// TIA Portal V17 export
// export: Created 2026-04-13T11:12:41.8044851Z, ExportSetting WithDefaults, DisplayName Totally Integrated Automation Portal, DisplayVersion V17 Update 4, DisplayName TIA Portal Openness, DisplayVersion V17 Update 4, DisplayName TIA Portal Version Control Interface, DisplayVersion V17, DisplayName SINAMICS Startdrive Advanced, DisplayVersion V17, DisplayName SINAMICS Startdrive G130, G150, S120, S150, SINAMICS MV, S210, DisplayVersion V17, DisplayName SINAMICS Startdrive G110M, G120, G120C, G120D, G120P, G115D, DisplayVersion V17, DisplayName STEP 7 Professional, DisplayVersion V17 Update 4, DisplayName STEP 7 Safety, DisplayVersion V17, DisplayName WinCC Professional, DisplayVersion V17 Update 4
FUNCTION_BLOCK "B1-开式保压"   // FB34, SCL
{ S7_Optimized_Access := 'TRUE' }
VERSION : 0.1
// stored: AutoNumber true, IsIECCheckEnabled false, IsRetainMemResEnabled false, MemoryReserve 100, SetENOAutomatically false, UDAEnableTagReadback false
   VAR_OUTPUT
      MBY等待保压 : Bool;
      MBY正在充气 : Bool;
      MBY保压不佳 : Bool;
      MBY正在保压 : Bool;
      MBY保压正常 : Bool;
   END_VAR
   VAR_IN_OUT
      模式设定 : Real;
      MBY保压 : Bool;
      MQT其他阀 : Bool;
      MCQ充气阀 : Bool;
      当前阶段 : Int;
      SV保压低设定 : Real;
      SV保压高设定 : Real;
      SV保压差值 : Real;
      SV保压时 : UInt;
      SV保压分 : UInt;
      SV保压秒 : UInt;
      PV塔内压力 { ExternalAccessible := 'False'; ExternalVisible := 'False'; ExternalWritable := 'False'} : Real;
      PV保压前 { ExternalAccessible := 'False'; ExternalVisible := 'False'; ExternalWritable := 'False'} : Real;
      PV保压后 { ExternalAccessible := 'False'; ExternalVisible := 'False'; ExternalWritable := 'False'} : Real;
      PV保压当前差值 { ExternalAccessible := 'False'; ExternalVisible := 'False'; ExternalWritable := 'False'} : Real;
      PV保压时 { ExternalAccessible := 'False'; ExternalVisible := 'False'; ExternalWritable := 'False'} : UInt;
      PV保压分 { ExternalAccessible := 'False'; ExternalVisible := 'False'; ExternalWritable := 'False'} : UInt;
      PV保压秒 { ExternalAccessible := 'False'; ExternalVisible := 'False'; ExternalWritable := 'False'} : UInt;
   END_VAR
   VAR
      T_1HZ { S7_SetPoint := 'True'} : TON_TIME;
   END_VAR
BEGIN
   IF #模式设定 = 3.0 OR #模式设定 = 4.0 THEN


       IF #MBY保压 THEN

           IF #当前阶段 = 5 THEN
               #当前阶段 := 1;
           END_IF;

      ELSE
           #当前阶段 := 5; 
       END_IF;

       (* IF #MCZ重置 THEN
           #当前阶段 := 4;
           #MCZ重置 := FALSE;

       END_IF;
       *)
       CASE #当前阶段 OF
           1://开始充气
               #MQT其他阀 := 0;
               #MCQ充气阀 := 1;
               #MBY等待保压 := 0;
               #MBY正在充气 := 1;
               #MBY保压不佳 := 0;
               #MBY正在保压 := 0;
               #MBY保压正常 := 0;

               IF (#PV塔内压力 >= #SV保压低设定) AND (#PV塔内压力 <= #SV保压高设定) THEN
                   #MCQ充气阀 := 0;
                   #PV保压前 := #PV塔内压力;
                   #当前阶段 := 2;
               END_IF;
           2://时间记录
               IF #T_1HZ.Q THEN
                   #PV保压秒 += 1;
                   IF #PV保压秒 >= 60 THEN
                       #PV保压分 += 1;
                       #PV保压秒 := 0;
                       IF #PV保压分 >= 60 THEN
                           #PV保压时 += 1;
                           #PV保压分 := 0;
                       END_IF;
                   END_IF;
               END_IF;
               IF (#PV保压时 > #SV保压时) OR ((#PV保压时 = #SV保压时) AND (#PV保压分 > #SV保压分)) OR ((#PV保压时 = #SV保压时) AND (#PV保压分 = #SV保压分) AND (#PV保压秒 >= #SV保压秒)) THEN
                   #PV保压后 := #PV塔内压力;
                   #当前阶段 := 3;
               END_IF;

               #MBY等待保压 := 0;
               #MBY正在充气 := 0;
               #MBY保压不佳 := 0;
               #MBY正在保压 := 1;
               #MBY保压正常 := 0;

           3://保压结束
               #PV保压当前差值 := ABS(#PV保压前 - #PV保压后);
               #MBY保压正常 := #PV保压当前差值 < #SV保压差值;
               #MBY保压不佳 := NOT (#PV保压当前差值 < #SV保压差值);
               IF #MBY保压正常 OR #MBY保压不佳 THEN
                   #MBY正在保压 := 0;
                   #当前阶段 :=4;
               END_IF;
           4://停止保压，并记录数据



               #MBY正在充气 := 0;

               #MBY正在保压 := 0;



           5://清空数据
               #MCQ充气阀 := 0;
               #MBY保压 := 0;
               #PV保压前 := 0;
               #PV保压后 := 0;
               #PV保压时 := 0;
               #PV保压分 := 0;
               #PV保压秒 := 0;


               #MBY等待保压 := 1;
               #MBY正在充气 := 0;

               #MBY正在保压 := 0;
               #MBY保压正常 := 0;
               #MBY保压不佳 := 0;

               #PV保压当前差值 := 0.0;
       END_CASE;

       #T_1HZ(IN := NOT #T_1HZ.Q,
              PT := T#1S);
   END_IF;
END_FUNCTION_BLOCK
